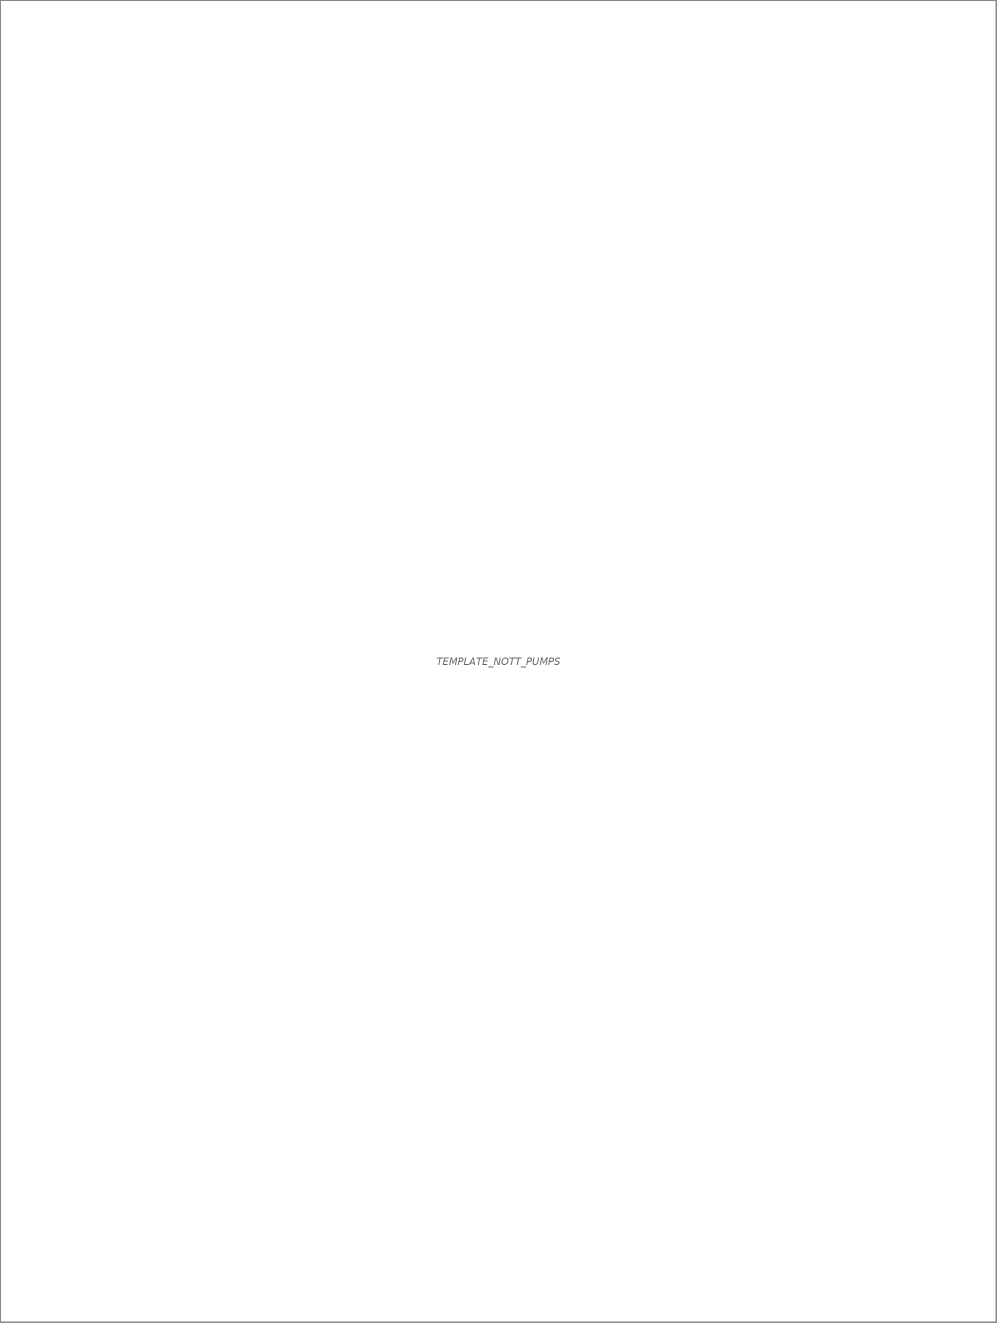
VISUALIZATION VISU_NOTT_RP  // 997x1323
    Frame (0,0 997x1323)
        shows TEMPLATE_NOTT_PUMPS(m_Instance := MAIN.nott_cryo_ctrl.evac.pump_pvp)
END_VISUALIZATION

(* stored: Version 1.1.0.1, ProductVersion 3.1.4026.18
   Visu VISU_NOTT_RP: Id {657b383a-1664-427c-8c32-bd9eb4ae2d2d} *)
